// TwinCAT 3 PLC project PLC
// Title: TcCoE
// Company: Roald
// Author: Roald
// ProjectVersion: 0.1.0
// Description: This library wraps `Tc2_EtherCAT.FB_EcCoESdoWriteEx` and `Tc2_EtherCAT.FB_EcCoESdoReadEx`, to have better error messages using the [TcError](https://github.com/Roald87/TcError/) library.
// ProgramVersion: 3.1.4023.0
// libraries:
//   Tc2_EtherCAT, * (Beckhoff Automation GmbH)
//   Tc2_Standard, * (Beckhoff Automation GmbH)
//   Tc2_System, * (Beckhoff Automation GmbH)
//   Tc3_Module, * (Beckhoff Automation GmbH)
//   TcError, * (Roald)
// project tree:
//   CoE/ AmsNetAddress.TcDUT, CoeReaderEx.TcPOU, CoeWriterEx.TcPOU, ProcessDataObjectIndex.TcDUT
//   / PlcTask.TcTTO

CONFIGURATION PLC
    RESOURCE PLC ON TwinCAT3
        TASK PlcTask(INTERVAL := T#10ms, PRIORITY := 20);
    END_RESOURCE
END_CONFIGURATION

// ---- CoE/AmsNetAddress.TcDUT
TYPE AmsNetAddress : STRUCT
    netId : Tc2_System.T_AmsNetID;
    port : T_AmsPort;
END_STRUCT
END_TYPE

// ---- CoE/ProcessDataObjectIndex.TcDUT
TYPE ProcessDataObjectIndex : STRUCT
    index : WORD;
    subIndex : BYTE;
END_STRUCT
END_TYPE

// ---- CoE/CoeReaderEx.TcPOU
FUNCTION_BLOCK CoeReaderEx EXTENDS FB_EcCoESdoReadEx
VAR_OUTPUT
    eAdsError : TcError.AdsErrorCodes;
END_VAR

SUPER^();
eAdsError := TcError.ToAdsErrorCode(SUPER^.nErrId);

END_FUNCTION_BLOCK

// ---- CoE/CoeWriterEx.TcPOU
FUNCTION_BLOCK CoeWriterEx
VAR_INPUT
    index : ProcessDataObjectIndex; (* CANopen Sdo index.*)
    pSrcBuf : PVOID; (* Contains the address of the buffer containing the data to be send. *)
    cbBufLen : UDINT; (* Contains the max. number of bytes to be received. *)
    bExecute : BOOL; (* Function block execution is triggered by a rising edge at this input.*)
    tTimeout : TIME := DEFAULT_ADS_TIMEOUT; (* States the time before the function is cancelled. *)
    bCompleteAccess : BOOL; (* access complete object*)
END_VAR
VAR_OUTPUT
    bBusy : BOOL;
    bError : BOOL;
    eAdsError : TcError.AdsErrorCodes;
END_VAR
VAR
    writer : Tc2_EtherCAT.FB_EcCoESdoWriteEx;
    _amsNetAddress : AmsNetAddress; (* AmsNetId of the EtherCAT master device.*)
END_VAR

writer(
    sNetId:=_amsNetAddress.netId,
    nSlaveAddr:=_amsNetAddress.port,
    nIndex:=index.index,
    nSubIndex:=index.subIndex,
    pSrcBuf:=pSrcBuf,
    cbBufLen:=cbBufLen,
    bExecute:=bExecute,
    tTimeout:=tTimeOut,
    bCompleteAccess:=bCompleteAccess,
    bBusy=>bBusy,
    bError=>bError,
);
eAdsError := TcError.ToAdsErrorCode(writer.nErrId);

METHOD FB_init : BOOL
VAR_INPUT
    bInitRetains : BOOL; // if TRUE, the retain variables are initialized (warm start / cold start)
    bInCopyCode :
        BOOL; // if TRUE, the instance afterwards gets moved into the copy code (online change)
    amsNetAddress : AmsNetAddress;
END_VAR
THIS^._amsNetAddress := amsNetAddress;
END_METHOD

END_FUNCTION_BLOCK
